FUNCTION_BLOCK ASR_SR_TO_2AE (* Composite FB for convert ASR to 2 AE *)
  (* Standard: 61499-2; Description: Copyright (c) 2026 HR Agrartechnik GmbH This program and the accompanying materials are made available under the terms of the Eclipse Public License 2.0 which is available at https://www.eclipse.org/legal/epl-2.0/ SPDX-License-Identifier: EPL-2.0 *)
  (* Version 1.0, 2026-09-06, Franz Höpfinger, HR Agrartechnik GmbH *)
  PACKAGE adapter::conversion::unidirectional;
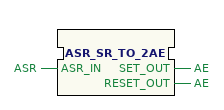
  SOCKETS
    ASR_IN : adapter::types::unidirectional::ASR; (* Adapter Input *)
  END_SOCKETS
  PLUGS
    SET_OUT : adapter::types::unidirectional::AE; (* Set / Switch on *)
    RESET_OUT : adapter::types::unidirectional::AE; (* Reset / Switch off *)
  END_PLUGS
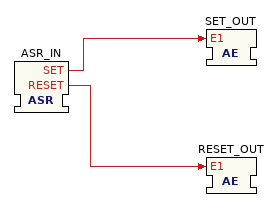
  EVENT_CONNECTIONS
    ASR_IN.SET TO SET_OUT.E1;
    ASR_IN.RESET TO RESET_OUT.E1;
  END_CONNECTIONS
END_FUNCTION_BLOCK
